// TIA Portal V19 export
TYPE "LAF_typeAlarms"
// Alarms of the module
// stored: Access Published
   STRUCT
      error : Bool;   // Error is active
      warning : Bool;   // Warning is active
      info : Bool;   // Info is active
   END_STRUCT;
END_TYPE
